LIN {X 0,Y 77.091,Z 1197.303,A -85,B 0,C 180,E1 -2217.871,E2 -2217.871} C_VEL
LIN {X 0,Y 72.704,Z 1199.365,A -85,B 0,C 180,E1 -2233.21,E2 -2233.21} C_VEL
LIN {X 0,Y 71.914,Z 1200.384,A -85,B 0,C 180,E1 -2246.011,E2 -2246.011} C_VEL
LIN {X 0,Y 71.92,Z 1200.628,A -85,B 0,C 180,E1 -2254.782,E2 -2254.782} C_VEL
LIN {X 0,Y 72.612,Z 1200.606,A -85,B 0,C 180,E1 -2265.983,E2 -2265.983} C_VEL
LIN {X 0,Y 76.855,Z 1199.806,A -85,B 0,C 180,E1 -2281.355,E2 -2281.355} C_VEL
LIN {X 0,Y 86.243,Z 1197.883,A -85,B 0,C 180,E1 -2295.953,E2 -2295.953} C_VEL
LIN {X 0,Y 99.626,Z 1194.884,A -85,B 0,C 180,E1 -2307.459,E2 -2307.459} C_VEL
LIN {X 0,Y 115.844,Z 1190.793,A -85,B 0,C 180,E1 -2316.188,E2 -2316.188} C_VEL
LIN {X 0,Y 137.433,Z 1184.57,A -85,B 0,C 180,E1 -2323.805,E2 -2323.805} C_VEL
LIN {X 0,Y 162.579,Z 1175.891,A -85,B 0,C 180,E1 -2329.732,E2 -2329.732} C_VEL
LIN {X 0,Y 183.237,Z 1167.701,A -85,B 0,C 180,E1 -2333.267,E2 -2333.267} C_VEL
LIN {X 0,Y 203.474,Z 1158.67,A -85,B 0,C 180,E1 -2335.969,E2 -2335.969} C_VEL
LIN {X 0,Y 215.208,Z 1152.962,A -85,B 0,C 180,E1 -2337.298,E2 -2337.298} C_VEL
LIN {X 0,Y 187.985,Z 1165.505,A -85,B 0,C 180,E1 -2340.671,E2 -2340.671} C_VEL
LIN {X 0,Y 166.767,Z 1173.941,A -85,B 0,C 180,E1 -2344.126,E2 -2344.126} C_VEL
LIN {X 0,Y 147.496,Z 1180.694,A -85,B 0,C 180,E1 -2348.227,E2 -2348.227} C_VEL
LIN {X 0,Y 127.742,Z 1186.76,A -85,B 0,C 180,E1 -2353.94,E2 -2353.94} C_VEL
LIN {X 0,Y 105.044,Z 1192.7,A -85,B 0,C 180,E1 -2363.971,E2 -2363.971} C_VEL
LIN {X 0,Y 88.975,Z 1196.171,A -85,B 0,C 180,E1 -2375.995,E2 -2375.995} C_VEL
LIN {X 0,Y 78.768,Z 1198.118,A -85,B 0,C 180,E1 -2389.659,E2 -2389.659} C_VEL
LIN {X 0,Y 73.501,Z 1198.999,A -85,B 0,C 180,E1 -2404.198,E2 -2404.198} C_VEL
LIN {X 0,Y 72.003,Z 1199.13,A -85,B 0,C 180,E1 -2417.166,E2 -2417.166} C_VEL
LIN {X 0,Y 71.917,Z 1198.846,A -85,B 0,C 180,E1 -2426.815,E2 -2426.815} C_VEL
LIN {X 0,Y 72.477,Z 1198.064,A -85,B 0,C 180,E1 -2437.933,E2 -2437.933} C_VEL
LIN {X 0,Y 75.642,Z 1196.495,A -85,B 0,C 180,E1 -2451.726,E2 -2451.726} C_VEL
LIN {X 0,Y 82.886,Z 1193.905,A -85,B 0,C 180,E1 -2465.386,E2 -2465.386} C_VEL
LIN {X 0,Y 94.12,Z 1190.203,A -85,B 0,C 180,E1 -2477.163,E2 -2477.163} C_VEL
LIN {X 0,Y 108.836,Z 1185.24,A -85,B 0,C 180,E1 -2486.725,E2 -2486.725} C_VEL
LIN {X 0,Y 127.287,Z 1178.53,A -85,B 0,C 180,E1 -2494.607,E2 -2494.607} C_VEL
LIN {X 0,Y 150.879,Z 1168.792,A -85,B 0,C 180,E1 -2501.385,E2 -2501.385} C_VEL
LIN {X 0,Y 170.467,Z 1159.639,A -85,B 0,C 180,E1 -2505.427,E2 -2505.427} C_VEL
LIN {X 0,Y 189.767,Z 1149.62,A -85,B 0,C 180,E1 -2508.534,E2 -2508.534} C_VEL
LIN {X 0,Y 211.404,Z 1137.13,A -85,B 0,C 180,E1 -2511.31,E2 -2511.31} C_VEL
LIN {X 0,Y 234.395,Z 1122.031,A -85,B 0,C 180,E1 -2513.687,E2 -2513.687} C_VEL
LIN {X 0,Y 252.832,Z 1108.504,A -85,B 0,C 180,E1 -2515.273,E2 -2515.273} C_VEL
LIN {X 0,Y 269.467,Z 1095.088,A -85,B 0,C 180,E1 -2516.519,E2 -2516.519} C_VEL
LIN {X 0,Y 274.052,Z 1091.217,A -85,B 0,C 180,E1 -2516.827,E2 -2516.827} C_VEL
LIN {X 0,Y 264.864,Z 1099.026,A -85,B 0,C 180,E1 -2517.452,E2 -2517.452} C_VEL
LIN {X 0,Y 258.902,Z 1103.925,A -85,B 0,C 180,E1 -2517.657,E2 -2517.657} C_VEL
LIN {X 0,Y 242.811,Z 1116.04,A -85,B 0,C 180,E1 -2517.44,E2 -2517.44} C_VEL
LIN {X 0,Y 236.54,Z 1120.44,A -85,B 0,C 180,E1 -2517.685,E2 -2517.685} C_VEL
LIN {X 0,Y 215.985,Z 1134.146,A -85,B 0,C 180,E1 -2519.492,E2 -2519.492} C_VEL
LIN {X 0,Y 191.123,Z 1148.746,A -85,B 0,C 180,E1 -2522.219,E2 -2522.219} C_VEL
LIN {X 0,Y 170.652,Z 1159.36,A -85,B 0,C 180,E1 -2525.077,E2 -2525.077} C_VEL
LIN {X 0,Y 151.639,Z 1168.21,A -85,B 0,C 180,E1 -2528.47,E2 -2528.47} C_VEL
LIN {X 0,Y 131.476,Z 1176.615,A -85,B 0,C 180,E1 -2533.228,E2 -2533.228} C_VEL
LIN {X 0,Y 107.54,Z 1185.351,A -85,B 0,C 180,E1 -2541.595,E2 -2541.595} C_VEL
LIN {X 0,Y 89.996,Z 1191.012,A -85,B 0,C 180,E1 -2551.479,E2 -2551.479} C_VEL
LIN {X 0,Y 77.165,Z 1194.95,A -85,B 0,C 180,E1 -2563.475,E2 -2563.475} C_VEL
LIN {X 0,Y 68.492,Z 1197.753,A -85,B 0,C 180,E1 -2578.291,E2 -2578.291} C_VEL
LIN {X 0,Y 64.574,Z 1199.459,A -85,B 0,C 180,E1 -2593.813,E2 -2593.813} C_VEL
LIN {X 0,Y 63.912,Z 1200.311,A -85,B 0,C 180,E1 -2606.409,E2 -2606.409} C_VEL
LIN {X 0,Y 63.942,Z 1200.552,A -85,B 0,C 180,E1 -2616.281,E2 -2616.281} C_VEL
LIN {X 0,Y 65.135,Z 1200.477,A -85,B 0,C 180,E1 -2629.734,E2 -2629.734} C_VEL
LIN {X 0,Y 70.613,Z 1199.625,A -85,B 0,C 180,E1 -2646.183,E2 -2646.183} C_VEL
LIN {X 0,Y 81.286,Z 1197.723,A -85,B 0,C 180,E1 -2660.795,E2 -2660.795} C_VEL
LIN {X 0,Y 96.134,Z 1194.698,A -85,B 0,C 180,E1 -2672.133,E2 -2672.133} C_VEL
LIN {X 0,Y 114.393,Z 1190.376,A -85,B 0,C 180,E1 -2680.728,E2 -2680.728} C_VEL
LIN {X 0,Y 138.96,Z 1183.495,A -85,B 0,C 180,E1 -2688.11,E2 -2688.11} C_VEL
LIN {X 0,Y 162.904,Z 1175.354,A -85,B 0,C 180,E1 -2692.949,E2 -2692.949} C_VEL
LIN {X 0,Y 183.417,Z 1167.38,A -85,B 0,C 180,E1 -2696.013,E2 -2696.013} C_VEL
LIN {X 0,Y 193.814,Z 1163.035,A -85,B 0,C 180,E1 -2697.324,E2 -2697.324} C_VEL
LIN {X 0,Y 167.994,Z 1173.29,A -85,B 0,C 180,E1 -2700.869,E2 -2700.869} C_VEL
LIN {X 0,Y 147.405,Z 1180.365,A -85,B 0,C 180,E1 -2704.669,E2 -2704.669} C_VEL
LIN {X 0,Y 127.755,Z 1186.228,A -85,B 0,C 180,E1 -2709.562,E2 -2709.562} C_VEL
LIN {X 0,Y 107.575,Z 1191.391,A -85,B 0,C 180,E1 -2716.802,E2 -2716.802} C_VEL
LIN {X 0,Y 85.463,Z 1196.002,A -85,B 0,C 180,E1 -2730.205,E2 -2730.205} C_VEL
LIN {X 0,Y 72.971,Z 1198.114,A -85,B 0,C 180,E1 -2744.564,E2 -2744.564} C_VEL
LIN {X 0,Y 66.085,Z 1199.08,A -85,B 0,C 180,E1 -2761.046,E2 -2761.046} C_VEL
LIN {X 0,Y 64.025,Z 1199.204,A -85,B 0,C 180,E1 -2776.456,E2 -2776.456} C_VEL
LIN {X 0,Y 63.92,Z 1198.921,A -85,B 0,C 180,E1 -2787.314,E2 -2787.314} C_VEL
LIN {X 0,Y 64.784,Z 1198.047,A -85,B 0,C 180,E1 -2800.677,E2 -2800.677} C_VEL
LIN {X 0,Y 69.203,Z 1196.299,A -85,B 0,C 180,E1 -2816.613,E2 -2816.613} C_VEL
LIN {X 0,Y 78.017,Z 1193.586,A -85,B 0,C 180,E1 -2830.873,E2 -2830.873} C_VEL
LIN {X 0,Y 91.472,Z 1189.58,A -85,B 0,C 180,E1 -2842.939,E2 -2842.939} C_VEL
LIN {X 0,Y 111.66,Z 1183.193,A -85,B 0,C 180,E1 -2853.572,E2 -2853.572} C_VEL
LIN {X 0,Y 133.431,Z 1175.16,A -85,B 0,C 180,E1 -2860.772,E2 -2860.772} C_VEL
LIN {X 0,Y 152.994,Z 1167.07,A -85,B 0,C 180,E1 -2865.299,E2 -2865.299} C_VEL
LIN {X 0,Y 172.322,Z 1158.126,A -85,B 0,C 180,E1 -2868.701,E2 -2868.701} C_VEL
LIN {X 0,Y 195.929,Z 1145.886,A -85,B 0,C 180,E1 -2871.911,E2 -2871.911} C_VEL
LIN {X 0,Y 219.03,Z 1132.024,A -85,B 0,C 180,E1 -2874.377,E2 -2874.377} C_VEL
LIN {X 0,Y 237.553,Z 1119.67,A -85,B 0,C 180,E1 -2875.996,E2 -2875.996} C_VEL
LIN {X 0,Y 248.152,Z 1112.1,A -85,B 0,C 180,E1 -2876.812,E2 -2876.812} C_VEL
LIN {X 0,Y 236.54,Z 1120.44,A -85,B 0,C 180,E1 -2877.685,E2 -2877.685} C_VEL
LIN {X 0,Y 230.21,Z 1124.901,A -85,B 0,C 180,E1 -2877.947,E2 -2877.947} C_VEL
LIN {X 0,Y 212.298,Z 1136.289,A -85,B 0,C 180,E1 -2877.805,E2 -2877.805} C_VEL
LIN {X 0,Y 206.652,Z 1139.55,A -85,B 0,C 180,E1 -2878.108,E2 -2878.108} C_VEL
LIN {X 0,Y 186.981,Z 1150.543,A -85,B 0,C 180,E1 -2880.13,E2 -2880.13} C_VEL
LIN {X 0,Y 167.162,Z 1160.481,A -85,B 0,C 180,E1 -2882.653,E2 -2882.653} C_VEL
LIN {X 0,Y 142.968,Z 1171.268,A -85,B 0,C 180,E1 -2886.72,E2 -2886.72} C_VEL
LIN {X 0,Y 118.821,Z 1180.368,A -85,B 0,C 180,E1 -2892.535,E2 -2892.535} C_VEL
LIN {X 0,Y 100.021,Z 1186.607,A -85,B 0,C 180,E1 -2899.262,E2 -2899.262} C_VEL
LIN {X 0,Y 83.134,Z 1191.633,A -85,B 0,C 180,E1 -2908.593,E2 -2908.593} C_VEL
LIN {X 0,Y 67.7,Z 1195.944,A -85,B 0,C 180,E1 -2923.636,E2 -2923.636} C_VEL
LIN {X 0,Y 57.937,Z 1198.921,A -85,B 0,C 180,E1 -2945.527,E2 -2945.527} C_VEL
LIN {X 0,Y 55.936,Z 1200.165,A -85,B 0,C 180,E1 -2963.839,E2 -2963.839} C_VEL
LIN {X 0,Y 55.913,Z 1200.391,A -85,B 0,C 180,E1 -2974.098,E2 -2974.098} C_VEL
LIN {X 0,Y 56.987,Z 1200.472,A -85,B 0,C 180,E1 -2989.469,E2 -2989.469} C_VEL
LIN {X 0,Y 63.715,Z 1199.629,A -85,B 0,C 180,E1 -3009.738,E2 -3009.738} C_VEL
LIN {X 0,Y 76.305,Z 1197.679,A -85,B 0,C 180,E1 -3025.637,E2 -3025.637} C_VEL
LIN {X 0,Y 92.523,Z 1194.674,A -85,B 0,C 180,E1 -3036.712,E2 -3036.712} C_VEL
LIN {X 0,Y 111.026,Z 1190.579,A -85,B 0,C 180,E1 -3044.49,E2 -3044.49} C_VEL
LIN {X 0,Y 134.663,Z 1184.349,A -85,B 0,C 180,E1 -3050.931,E2 -3050.931} C_VEL
LIN {X 0,Y 160.951,Z 1175.824,A -85,B 0,C 180,E1 -3055.725,E2 -3055.725} C_VEL
LIN {X 0,Y 172.292,Z 1171.749,A -85,B 0,C 180,E1 -3057.339,E2 -3057.339} C_VEL
LIN {X 0,Y 147.598,Z 1180.123,A -85,B 0,C 180,E1 -3061.165,E2 -3061.165} C_VEL
LIN {X 0,Y 127.555,Z 1185.952,A -85,B 0,C 180,E1 -3065.443,E2 -3065.443} C_VEL
LIN {X 0,Y 108.075,Z 1190.772,A -85,B 0,C 180,E1 -3071.291,E2 -3071.291} C_VEL
LIN {X 0,Y 87.704,Z 1194.973,A -85,B 0,C 180,E1 -3080.804,E2 -3080.804} C_VEL
LIN {X 0,Y 68.361,Z 1198.047,A -85,B 0,C 180,E1 -3097.903,E2 -3097.903} C_VEL
LIN {X 0,Y 59.196,Z 1199.141,A -85,B 0,C 180,E1 -3116.128,E2 -3116.128} C_VEL
LIN {X 0,Y 56.11,Z 1199.304,A -85,B 0,C 180,E1 -3134.501,E2 -3134.501} C_VEL
LIN {X 0,Y 55.909,Z 1199.041,A -85,B 0,C 180,E1 -3145.902,E2 -3145.902} C_VEL
LIN {X 0,Y 56.537,Z 1198.364,A -85,B 0,C 180,E1 -3159.163,E2 -3159.163} C_VEL
LIN {X 0,Y 60.629,Z 1196.88,A -85,B 0,C 180,E1 -3176.445,E2 -3176.445} C_VEL
LIN {X 0,Y 70.32,Z 1194.221,A -85,B 0,C 180,E1 -3193.044,E2 -3193.044} C_VEL
LIN {X 0,Y 84.627,Z 1190.364,A -85,B 0,C 180,E1 -3205.802,E2 -3205.802} C_VEL
LIN {X 0,Y 101.636,Z 1185.39,A -85,B 0,C 180,E1 -3214.839,E2 -3214.839} C_VEL
LIN {X 0,Y 122.952,Z 1178.376,A -85,B 0,C 180,E1 -3222.083,E2 -3222.083} C_VEL
LIN {X 0,Y 147.413,Z 1168.92,A -85,B 0,C 180,E1 -3227.621,E2 -3227.621} C_VEL
LIN {X 0,Y 168.058,Z 1159.76,A -85,B 0,C 180,E1 -3230.987,E2 -3230.987} C_VEL
LIN {X 0,Y 187.208,Z 1150.238,A -85,B 0,C 180,E1 -3233.434,E2 -3233.434} C_VEL
LIN {X 0,Y 207.606,Z 1138.921,A -85,B 0,C 180,E1 -3235.539,E2 -3235.539} C_VEL
LIN {X 0,Y 221.787,Z 1130.228,A -85,B 0,C 180,E1 -3236.801,E2 -3236.801} C_VEL
LIN {X 0,Y 206.652,Z 1139.55,A -85,B 0,C 180,E1 -3238.108,E2 -3238.108} C_VEL
LIN {X 0,Y 200.002,Z 1143.399,A -85,B 0,C 180,E1 -3238.454,E2 -3238.454} C_VEL
LIN {X 0,Y 181.276,Z 1153.406,A -85,B 0,C 180,E1 -3238.394,E2 -3238.394} C_VEL
LIN {X 0,Y 175.377,Z 1156.259,A -85,B 0,C 180,E1 -3238.772,E2 -3238.772} C_VEL
LIN {X 0,Y 152.057,Z 1166.844,A -85,B 0,C 180,E1 -3241.767,E2 -3241.767} C_VEL
LIN {X 0,Y 131.938,Z 1174.892,A -85,B 0,C 180,E1 -3245.218,E2 -3245.218} C_VEL
LIN {X 0,Y 111.687,Z 1182.014,A -85,B 0,C 180,E1 -3250.002,E2 -3250.002} C_VEL
LIN {X 0,Y 87.683,Z 1189.327,A -85,B 0,C 180,E1 -3258.824,E2 -3258.824} C_VEL
LIN {X 0,Y 67.971,Z 1194.362,A -85,B 0,C 180,E1 -3271.977,E2 -3271.977} C_VEL
LIN {X 0,Y 55.642,Z 1197.363,A -85,B 0,C 180,E1 -3288.322,E2 -3288.322} C_VEL
LIN {X 0,Y 49.367,Z 1199.156,A -85,B 0,C 180,E1 -3307.362,E2 -3307.362} C_VEL
LIN {X 0,Y 47.916,Z 1200.117,A -85,B 0,C 180,E1 -3325.207,E2 -3325.207} C_VEL
LIN {X 0,Y 47.933,Z 1200.316,A -85,B 0,C 180,E1 -3335.982,E2 -3335.982} C_VEL
LIN {X 0,Y 49.612,Z 1200.367,A -85,B 0,C 180,E1 -3353.766,E2 -3353.766} C_VEL
LIN {X 0,Y 57.755,Z 1199.549,A -85,B 0,C 180,E1 -3375.214,E2 -3375.214} C_VEL
LIN {X 0,Y 71.938,Z 1197.637,A -85,B 0,C 180,E1 -3391.114,E2 -3391.114} C_VEL
LIN {X 0,Y 89.548,Z 1194.651,A -85,B 0,C 180,E1 -3401.631,E2 -3401.631} C_VEL
LIN {X 0,Y 109.082,Z 1190.575,A -85,B 0,C 180,E1 -3408.741,E2 -3408.741} C_VEL
LIN {X 0,Y 132.634,Z 1184.62,A -85,B 0,C 180,E1 -3414.304,E2 -3414.304} C_VEL
LIN {X 0,Y 150.652,Z 1179.186,A -85,B 0,C 180,E1 -3417.337,E2 -3417.337} C_VEL
LIN {X 0,Y 127.924,Z 1185.698,A -85,B 0,C 180,E1 -3421.344,E2 -3421.344} C_VEL
LIN {X 0,Y 107.661,Z 1190.566,A -85,B 0,C 180,E1 -3426.435,E2 -3426.435} C_VEL
LIN {X 0,Y 87.614,Z 1194.517,A -85,B 0,C 180,E1 -3434.069,E2 -3434.069} C_VEL
LIN {X 0,Y 66.916,Z 1197.757,A -85,B 0,C 180,E1 -3448.173,E2 -3448.173} C_VEL
LIN {X 0,Y 52.829,Z 1199.202,A -85,B 0,C 180,E1 -3469.952,E2 -3469.952} C_VEL
LIN {X 0,Y 48.26,Z 1199.403,A -85,B 0,C 180,E1 -3491.899,E2 -3491.899} C_VEL
LIN {X 0,Y 47.907,Z 1199.138,A -85,B 0,C 180,E1 -3505.216,E2 -3505.216} C_VEL
LIN {X 0,Y 48.519,Z 1198.548,A -85,B 0,C 180,E1 -3519.494,E2 -3519.494} C_VEL
LIN {X 0,Y 53.542,Z 1197.017,A -85,B 0,C 180,E1 -3540.284,E2 -3540.284} C_VEL
LIN {X 0,Y 64.64,Z 1194.378,A -85,B 0,C 180,E1 -3557.948,E2 -3557.948} C_VEL
LIN {X 0,Y 80.341,Z 1190.541,A -85,B 0,C 180,E1 -3570.602,E2 -3570.602} C_VEL
LIN {X 0,Y 97.589,Z 1185.836,A -85,B 0,C 180,E1 -3578.813,E2 -3578.813} C_VEL
LIN {X 0,Y 117.046,Z 1179.78,A -85,B 0,C 180,E1 -3584.871,E2 -3584.871} C_VEL
LIN {X 0,Y 142.093,Z 1170.769,A -85,B 0,C 180,E1 -3590.122,E2 -3590.122} C_VEL
LIN {X 0,Y 166.007,Z 1160.495,A -85,B 0,C 180,E1 -3593.634,E2 -3593.634} C_VEL
LIN {X 0,Y 186.451,Z 1150.547,A -85,B 0,C 180,E1 -3595.926,E2 -3595.926} C_VEL
LIN {X 0,Y 195.288,Z 1145.996,A -85,B 0,C 180,E1 -3596.777,E2 -3596.777} C_VEL
LIN {X 0,Y 175.377,Z 1156.259,A -85,B 0,C 180,E1 -3598.772,E2 -3598.772} C_VEL
LIN {X 0,Y 168.413,Z 1159.533,A -85,B 0,C 180,E1 -3599.214,E2 -3599.214} C_VEL
LIN {X 0,Y 149.928,Z 1167.515,A -85,B 0,C 180,E1 -3599.245,E2 -3599.245} C_VEL
LIN {X 0,Y 142.887,Z 1170.36,A -85,B 0,C 180,E1 -3599.803,E2 -3599.803} C_VEL
LIN {X 0,Y 116.33,Z 1179.923,A -85,B 0,C 180,E1 -3604.391,E2 -3604.391} C_VEL
LIN {X 0,Y 95.4,Z 1186.318,A -85,B 0,C 180,E1 -3609.855,E2 -3609.855} C_VEL
LIN {X 0,Y 76.549,Z 1191.274,A -85,B 0,C 180,E1 -3617.528,E2 -3617.528} C_VEL
LIN {X 0,Y 58.953,Z 1195.3,A -85,B 0,C 180,E1 -3630.112,E2 -3630.112} C_VEL
LIN {X 0,Y 43.97,Z 1198.614,A -85,B 0,C 180,E1 -3655.348,E2 -3655.348} C_VEL
LIN {X 0,Y 39.99,Z 1199.947,A -85,B 0,C 180,E1 -3681.366,E2 -3681.366} C_VEL
LIN {X 0,Y 39.913,Z 1200.176,A -85,B 0,C 180,E1 -3694.305,E2 -3694.305} C_VEL
LIN {X 0,Y 41.721,Z 1200.337,A -85,B 0,C 180,E1 -3715.55,E2 -3715.55} C_VEL
LIN {X 0,Y 52.27,Z 1199.488,A -85,B 0,C 180,E1 -3741.648,E2 -3741.648} C_VEL
LIN {X 0,Y 68.308,Z 1197.594,A -85,B 0,C 180,E1 -3757.238,E2 -3757.238} C_VEL
LIN {X 0,Y 87.275,Z 1194.627,A -85,B 0,C 180,E1 -3766.848,E2 -3766.848} C_VEL
LIN {X 0,Y 107.759,Z 1190.572,A -85,B 0,C 180,E1 -3773.119,E2 -3773.119} C_VEL
LIN {X 0,Y 128.412,Z 1185.578,A -85,B 0,C 180,E1 -3777.38,E2 -3777.38} C_VEL
LIN {X 0,Y 107.036,Z 1190.567,A -85,B 0,C 180,E1 -3781.817,E2 -3781.817} C_VEL
LIN {X 0,Y 86.854,Z 1194.38,A -85,B 0,C 180,E1 -3788.111,E2 -3788.111} C_VEL
LIN {X 0,Y 65.739,Z 1197.463,A -85,B 0,C 180,E1 -3799.447,E2 -3799.447} C_VEL
LIN {X 0,Y 47.214,Z 1199.264,A -85,B 0,C 180,E1 -3822.172,E2 -3822.172} C_VEL
LIN {X 0,Y 40.526,Z 1199.503,A -85,B 0,C 180,E1 -3848.285,E2 -3848.285} C_VEL
LIN {X 0,Y 39.907,Z 1199.213,A -85,B 0,C 180,E1 -3865.695,E2 -3865.695} C_VEL
LIN {X 0,Y 40.802,Z 1198.597,A -85,B 0,C 180,E1 -3882.747,E2 -3882.747} C_VEL
LIN {X 0,Y 47.258,Z 1197.042,A -85,B 0,C 180,E1 -3906.335,E2 -3906.335} C_VEL
LIN {X 0,Y 60.395,Z 1194.343,A -85,B 0,C 180,E1 -3924.588,E2 -3924.588} C_VEL
LIN {X 0,Y 77.516,Z 1190.516,A -85,B 0,C 180,E1 -3936.331,E2 -3936.331} C_VEL
LIN {X 0,Y 96.751,Z 1185.536,A -85,B 0,C 180,E1 -3943.977,E2 -3943.977} C_VEL
LIN {X 0,Y 119.89,Z 1178.517,A -85,B 0,C 180,E1 -3949.783,E2 -3949.783} C_VEL
LIN {X 0,Y 145.921,Z 1168.983,A -85,B 0,C 180,E1 -3954.1,E2 -3954.1} C_VEL
LIN {X 0,Y 167.267,Z 1159.881,A -85,B 0,C 180,E1 -3956.658,E2 -3956.658} C_VEL
LIN {X 0,Y 168.017,Z 1159.539,A -85,B 0,C 180,E1 -3956.768,E2 -3956.768} C_VEL
LIN {X 0,Y 146.998,Z 1168.656,A -85,B 0,C 180,E1 -3959.231,E2 -3959.231} C_VEL
LIN {X 0,Y 142.887,Z 1170.36,A -85,B 0,C 180,E1 -3959.803,E2 -3959.803} C_VEL
LIN {X 0,Y 135.788,Z 1173.125,A -85,B 0,C 180,E1 -3960.417,E2 -3960.417} C_VEL
LIN {X 0,Y 115.621,Z 1179.85,A -85,B 0,C 180,E1 -3960.69,E2 -3960.69} C_VEL
LIN {X 0,Y 109.414,Z 1181.759,A -85,B 0,C 180,E1 -3961.437,E2 -3961.437} C_VEL
LIN {X 0,Y 83.788,Z 1188.967,A -85,B 0,C 180,E1 -3967.899,E2 -3967.899} C_VEL
LIN {X 0,Y 60.249,Z 1194.153,A -85,B 0,C 180,E1 -3978.913,E2 -3978.913} C_VEL
LIN {X 0,Y 44.007,Z 1197.204,A -85,B 0,C 180,E1 -3995.112,E2 -3995.112} C_VEL
LIN {X 0,Y 34.522,Z 1198.992,A -85,B 0,C 180,E1 -4018.57,E2 -4018.57} C_VEL
LIN {X 0,Y 31.919,Z 1199.946,A -85,B 0,C 180,E1 -4044.601,E2 -4044.601} C_VEL
LIN {X 0,Y 32.059,Z 1200.142,A -85,B 0,C 180,E1 -4060.778,E2 -4060.778} C_VEL
LIN {X 0,Y 36.6,Z 1200.131,A -85,B 0,C 180,E1 -4088.919,E2 -4088.919} C_VEL
LIN {X 0,Y 49.827,Z 1199.214,A -85,B 0,C 180,E1 -4111.989,E2 -4111.989} C_VEL
LIN {X 0,Y 68.203,Z 1197.204,A -85,B 0,C 180,E1 -4125.358,E2 -4125.358} C_VEL
LIN {X 0,Y 88.617,Z 1194.12,A -85,B 0,C 180,E1 -4133.155,E2 -4133.155} C_VEL
LIN {X 0,Y 105.903,Z 1190.814,A -85,B 0,C 180,E1 -4137.416,E2 -4137.416} C_VEL
LIN {X 0,Y 83.127,Z 1194.88,A -85,B 0,C 180,E1 -4143.348,E2 -4143.348} C_VEL
LIN {X 0,Y 57.272,Z 1198.166,A -85,B 0,C 180,E1 -4156.231,E2 -4156.231} C_VEL
LIN {X 0,Y 40.152,Z 1199.407,A -85,B 0,C 180,E1 -4177.177,E2 -4177.177} C_VEL
LIN {X 0,Y 32.604,Z 1199.553,A -85,B 0,C 180,E1 -4206.512,E2 -4206.512} C_VEL
LIN {X 0,Y 31.908,Z 1199.287,A -85,B 0,C 180,E1 -4226.414,E2 -4226.414} C_VEL
LIN {X 0,Y 33.267,Z 1198.647,A -85,B 0,C 180,E1 -4247.498,E2 -4247.498} C_VEL
LIN {X 0,Y 41.642,Z 1197.068,A -85,B 0,C 180,E1 -4274.141,E2 -4274.141} C_VEL
LIN {X 0,Y 56.711,Z 1194.379,A -85,B 0,C 180,E1 -4291.838,E2 -4291.838} C_VEL
LIN {X 0,Y 74.624,Z 1190.693,A -85,B 0,C 180,E1 -4302.059,E2 -4302.059} C_VEL
LIN {X 0,Y 94.825,Z 1185.734,A -85,B 0,C 180,E1 -4308.715,E2 -4308.715} C_VEL
LIN {X 0,Y 117.745,Z 1179.032,A -85,B 0,C 180,E1 -4313.503,E2 -4313.503} C_VEL
LIN {X 0,Y 140.358,Z 1171.228,A -85,B 0,C 180,E1 -4316.745,E2 -4316.745} C_VEL
LIN {X 0,Y 114.445,Z 1180.183,A -85,B 0,C 180,E1 -4320.501,E2 -4320.501} C_VEL
LIN {X 0,Y 109.414,Z 1181.759,A -85,B 0,C 180,E1 -4321.437,E2 -4321.437} C_VEL
LIN {X 0,Y 102.151,Z 1183.98,A -85,B 0,C 180,E1 -4322.352,E2 -4322.352} C_VEL
LIN {X 0,Y 81.023,Z 1189.26,A -85,B 0,C 180,E1 -4323.162,E2 -4323.162} C_VEL
LIN {X 0,Y 75.25,Z 1190.48,A -85,B 0,C 180,E1 -4324.312,E2 -4324.312} C_VEL
LIN {X 0,Y 55.331,Z 1194.489,A -85,B 0,C 180,E1 -4332.606,E2 -4332.606} C_VEL
LIN {X 0,Y 38.27,Z 1197.301,A -85,B 0,C 180,E1 -4347.324,E2 -4347.324} C_VEL
LIN {X 0,Y 26.96,Z 1199.015,A -85,B 0,C 180,E1 -4373.591,E2 -4373.591} C_VEL
LIN {X 0,Y 23.911,Z 1199.873,A -85,B 0,C 180,E1 -4405.193,E2 -4405.193} C_VEL
LIN {X 0,Y 24.318,Z 1200.065,A -85,B 0,C 180,E1 -4426.718,E2 -4426.718} C_VEL
LIN {X 0,Y 31.48,Z 1200.018,A -85,B 0,C 180,E1 -4460.562,E2 -4460.562} C_VEL
LIN {X 0,Y 47.38,Z 1199.082,A -85,B 0,C 180,E1 -4481.726,E2 -4481.726} C_VEL
LIN {X 0,Y 67.538,Z 1197.045,A -85,B 0,C 180,E1 -4492.68,E2 -4492.68} C_VEL
LIN {X 0,Y 82.76,Z 1194.951,A -85,B 0,C 180,E1 -4497.467,E2 -4497.467} C_VEL
LIN {X 0,Y 55.492,Z 1198.23,A -85,B 0,C 180,E1 -4507.717,E2 -4507.717} C_VEL
LIN {X 0,Y 34.956,Z 1199.509,A -85,B 0,C 180,E1 -4527.55,E2 -4527.55} C_VEL
LIN {X 0,Y 24.978,Z 1199.628,A -85,B 0,C 180,E1 -4561.301,E2 -4561.301} C_VEL
LIN {X 0,Y 23.903,Z 1199.384,A -85,B 0,C 180,E1 -4585.21,E2 -4585.21} C_VEL
LIN {X 0,Y 25.421,Z 1198.83,A -85,B 0,C 180,E1 -4610.741,E2 -4610.741} C_VEL
LIN {X 0,Y 36.291,Z 1197.204,A -85,B 0,C 180,E1 -4643.045,E2 -4643.045} C_VEL
LIN {X 0,Y 53.367,Z 1194.535,A -85,B 0,C 180,E1 -4659.53,E2 -4659.53} C_VEL
LIN {X 0,Y 73.472,Z 1190.668,A -85,B 0,C 180,E1 -4668.49,E2 -4668.49} C_VEL
LIN {X 0,Y 94.543,Z 1185.683,A -85,B 0,C 180,E1 -4673.809,E2 -4673.809} C_VEL
LIN {X 0,Y 111.539,Z 1180.921,A -85,B 0,C 180,E1 -4676.722,E2 -4676.722} C_VEL
LIN {X 0,Y 89.468,Z 1187.101,A -85,B 0,C 180,E1 -4680.64,E2 -4680.64} C_VEL
LIN {X 0,Y 75.25,Z 1190.48,A -85,B 0,C 180,E1 -4684.312,E2 -4684.312} C_VEL
LIN {X 0,Y 67.894,Z 1192.063,A -85,B 0,C 180,E1 -4685.88,E2 -4685.88} C_VEL
LIN {X 0,Y 46.5,Z 1195.691,A -85,B 0,C 180,E1 -4688.303,E2 -4688.303} C_VEL
LIN {X 0,Y 40.758,Z 1196.455,A -85,B 0,C 180,E1 -4690.914,E2 -4690.914} C_VEL
LIN {X 0,Y 22.28,Z 1198.757,A -85,B 0,C 180,E1 -4716.101,E2 -4716.101} C_VEL
LIN {X 0,Y 15.93,Z 1199.776,A -85,B 0,C 180,E1 -4762.774,E2 -4762.774} C_VEL
LIN {X 0,Y 16.481,Z 1199.947,A -85,B 0,C 180,E1 -4791.332,E2 -4791.332} C_VEL
LIN {X 0,Y 26.312,Z 1199.96,A -85,B 0,C 180,E1 -4832.87,E2 -4832.87} C_VEL
LIN {X 0,Y 45.467,Z 1199.02,A -85,B 0,C 180,E1 -4851.694,E2 -4851.694} C_VEL
LIN {X 0,Y 58.749,Z 1197.961,A -85,B 0,C 180,E1 -4857.501,E2 -4857.501} C_VEL
LIN {X 0,Y 32.831,Z 1199.572,A -85,B 0,C 180,E1 -4872.982,E2 -4872.982} C_VEL
LIN {X 0,Y 18.166,Z 1199.729,A -85,B 0,C 180,E1 -4908.678,E2 -4908.678} C_VEL
LIN {X 0,Y 15.903,Z 1199.458,A -85,B 0,C 180,E1 -4946.409,E2 -4946.409} C_VEL
LIN {X 0,Y 19.115,Z 1198.813,A -85,B 0,C 180,E1 -4985.141,E2 -4985.141} C_VEL
LIN {X 0,Y 32.949,Z 1197.229,A -85,B 0,C 180,E1 -5015.575,E2 -5015.575} C_VEL
LIN {X 0,Y 52.046,Z 1194.536,A -85,B 0,C 180,E1 -5028.481,E2 -5028.481} C_VEL
LIN {X 0,Y 73.269,Z 1190.643,A -85,B 0,C 180,E1 -5035.044,E2 -5035.044} C_VEL
LIN {X 0,Y 81.126,Z 1189.032,A -85,B 0,C 180,E1 -5036.722,E2 -5036.722} C_VEL
LIN {X 0,Y 56.085,Z 1194,A -85,B 0,C 180,E1 -5043.218,E2 -5043.218} C_VEL
LIN {X 0,Y 40.758,Z 1196.455,A -85,B 0,C 180,E1 -5050.914,E2 -5050.914} C_VEL
LIN {X 0,Y 33.533,Z 1197.357,A -85,B 0,C 180,E1 -5055.096,E2 -5055.096} C_VEL
LIN {X 0,Y 20,Z 1198.696,A -85,B 0,C 180,E1 -5062.588,E2 -5062.588} C_VEL
LIN {X 0,Y 10.219,Z 1199.406,A -85,B 0,C 180,E1 -5084.713,E2 -5084.713} C_VEL
LIN {X 0,Y 8.713,Z 1199.586,A -85,B 0,C 180,E1 -5099.068,E2 -5099.068} C_VEL
LIN {X 0,Y 8.03,Z 1199.767,A -85,B 0,C 180,E1 -5144.392,E2 -5144.392} C_VEL
LIN {X 0,Y 20.509,Z 1199.967,A -85,B 0,C 180,E1 -5207.134,E2 -5207.134} C_VEL
LIN {X 0,Y 32.774,Z 1199.639,A -85,B 0,C 180,E1 -5217.612,E2 -5217.612} C_VEL
LIN {X 0,Y 12.348,Z 1199.804,A -85,B 0,C 180,E1 -5247.08,E2 -5247.08} C_VEL
LIN {X 0,Y 7.92,Z 1199.533,A -85,B 0,C 180,E1 -5310.028,E2 -5310.028} C_VEL
LIN {X 0,Y 15.828,Z 1198.73,A -85,B 0,C 180,E1 -5372.208,E2 -5372.208} C_VEL
LIN {X 0,Y 33.399,Z 1197.033,A -85,B 0,C 180,E1 -5391.132,E2 -5391.132} C_VEL
LIN {X 0,Y 47.793,Z 1195.206,A -85,B 0,C 180,E1 -5396.698,E2 -5396.698} C_VEL
LIN {X 0,Y 21.431,Z 1198.427,A -85,B 0,C 180,E1 -5411.488,E2 -5411.488} C_VEL
LIN {X 0,Y 8.713,Z 1199.586,A -85,B 0,C 180,E1 -5459.068,E2 -5459.068} C_VEL
LIN {X 0,Y 8.177,Z 1201.582,A -85,B 0,C 180,E1 -5471.229,E2 -5471.229} C_VEL
LIN {X 0,Y 8.177,Z 1215,A -85,B 0,C 180,E1 -5471.229,E2 -5471.229} C_VEL
LIN {X 0,Y 8.177,Z 1215,A -85,B 0,C 180,E1 -5471.229,E2 -5471.229}

QRS_NEXT_CUT()

QRS_NEXT()
QRS_HOME()

END
